// TwinCAT 3 PLC project PLC
// ProgramVersion: 3.1.4024.0
// libraries:
//   Tc2_EtherCAT, * (Beckhoff Automation GmbH)
//   Tc2_MC2, * (Beckhoff Automation GmbH)
//   Tc2_NC, * (Beckhoff Automation GmbH)
//   Tc2_Standard, * (Beckhoff Automation GmbH)
//   Tc2_System, * (Beckhoff Automation GmbH)
//   Tc2_Utilities, * (Beckhoff Automation GmbH)
//   Tc3_Module, * (Beckhoff Automation GmbH)
// project tree:
//   DUTs/EtherCAT_Diag/ E_EcDiacStatus.TcDUT, E_EcGetSlaveName.TcDUT, E_EcSystemStatus.TcDUT, ST_EcTerminalDiagInfo.TcDUT
//   DUTs/TwinSAFE_Diag/ ST_AdsAddr.TcDUT
//   DUTs/TwinSAFE_Diag/TwinSAFE_Connection/EL1904/ ST_TsConnectionInfoEL1904.TcDUT, ST_TsDiagObjectsBitsEL1904.TcDUT, ST_TsDiagObjectsEL1904.TcDUT, ST_TsSlaveInfoEL1904.TcDUT
//   DUTs/TwinSAFE_Diag/TwinSAFE_Connection/EL2904/ ST_TsConnectionInfoEL2904.TcDUT, ST_TsDiagObjectsBitsEL2904.TcDUT, ST_TsDiagObjectsEL2904.TcDUT, ST_TsSlaveInfoEL2904.TcDUT
//   DUTs/TwinSAFE_Diag/TwinSAFE_Connection/EL6910/ ST_TsDeviceInfoDataC.TcDUT, ST_TsSlaveInfoEL6910.TcDUT
//   DUTs/TwinSAFE_Diag/TwinSAFE_Connection/ E_TsCycleDiagObj.TcDUT, ST_TsConnectionInfo12Byte.TcDUT, ST_TsConnectionInfo1Byte.TcDUT, ST_TsConnectionInfo2Byte.TcDUT, ST_TsConnectionInfo4Byte.TcDUT, ST_TsConnectionInfo8Byte.TcDUT, ST_TsSlave2Temp.TcDUT, ST_TsSlave3Temp.TcDUT, ST_TsSlaveAddress.TcDUT, ST_TsSlaveAddressCRC.TcDUT
//   DUTs/TwinSAFE_Diag/TwinSAFE_Functionblocks/ E_TsFbType.TcDUT, ST_TsFbInfo.TcDUT
//   DUTs/TwinSAFE_Diag/TwinSAFE_Group/ ST_TsGroupInfo.TcDUT
//   GVLs/ IO.TcGVL
//   / PlcTask.TcTTO
//   POUs/ FB_EcGetSlaveName.TcPOU (not stored), FB_TwinSafeConnectionEL1904.TcPOU, FB_TwinSafeConnectionEL2904.TcPOU (not stored), FB_TwinSafeConnectionEL6910.TcPOU (not stored), FB_TwinSafeFB.TcPOU, FB_TwinSafeGroup.TcPOU, FB_TwinSafeGroupExt.TcPOU, F_Scale.TcPOU, MAIN.TcPOU, PRG_Safety.TcPOU
// real-time tasks:
//   TASK PlcTask: cycle T#10ms, priority 20, ADS port 350
// motion (NC):
//   TASK NC-Task 1 SAF: cycle T#2ms, priority 4, ADS port 501
//   TASK NC-Task 1 SVB: cycle T#10ms, priority 8, ADS port 511
//   AXIS Axis 1 (id 1)
//     OtherSettings: AllowMotionCmdToSlave=true
//     encoder EncType=4
//       EncPara: MaxCount=#x0000ffff
//         Inc: RefSoftSyncMask=#x0000ffff
//     drive DrvType=24
//       Analog: TorqueSetpointScale=10, ScaleFactorActTorque=0.1
//       TimeComp: TaskDelayCycles=1
//     controller CtrType=1
//       CtrPara: PriorControlFactor=1
//         Observer: BandWidth=20
//   AXIS Axis 2 (id 2)
//     Dynamic: Acceleration=12727.1, Deceleration=12727.1, Jerk=38181.3
//     Velo: RefSearch=84.8472746666667, RefSync=84.8472746666667, SlowManual=424.236373333333, FastManual=2545.41824, Fast=8484.72746666667, Maximum=8484.73
//     OtherSettings: AllowMotionCmdToSlave=true
//     encoder EncType=19
//       EncPara: ScaleFactorNumerator=104.8576, ScaleFactorDenominator=1048576, MaxCount=#xffffffff
//     drive DrvType=16
//       DrvPara: MaxCount=#xffffffff, DriveControlDWord=#x00020000
//         Analog: VeloReferenz=9333.20021333334, VeloScale=32, TorqueSetpointScale=10, ScaleFactorActTorque=0.1
//         TimeComp: TaskDelayCycles=1
//     controller CtrType=1
//       CtrPara: PriorControlFactor=1
//         PosDiffControl: Enable=false
//         Observer: BandWidth=20
// I/O:
//   DEVICE Device 1 (EtherCAT), AmsNetId 5.71.184.138.2.1
//     Term 1 (EK1200) [EK1200-5000 EtherCAT Power supply (2A E-Bus)]
//       Term 2 (EL1014) [EL1014 4Ch. Dig. Input 24V, 10µs]
//       Term 3 (EL2014) [EL2014 4Ch. Dig. Output 24V, 0,5A, Diagnostic]
//       Term 4 (EL6910) [EL6910, TwinSAFE PLC]
//       Term 5 (EL1904) [EL1904, 4 Ch. Safety Input 24V, TwinSAFE]
//         modules: Module 1 (FSOES)
//       Term 6 (EL3102) [EL3102 2Ch. Ana. Input +/-10V, Diff.]
//       Term 7 (EL9512) [EL9512 Power supply terminal 12V]
//       Term 8 (EK1122) [EK1122 2 port EtherCAT junction]
//         Term 9 (EK1818) [EK1818 EtherCAT IO-Coupler  (1A E-Bus, 8 Ch. Dig. In, 3ms, 4 Ch. Dig. Out 24V, 0,5A)]
//           Term 10 (EL1809) [EL1809 16Ch. Dig. Input 24V, 3ms]
//           Term 11 (EL2809) [EL2809 16Ch. Dig. Output 24V, 0.5A]
//           Term 12 (EL2904) [EL2904, 4 Ch. Safety Output 24V, 0.5A, TwinSAFE]
//             modules: Module 1 (FSOES), Module 2 (DO)
//           Term 13 (EL9110) [EL9110 Power Supplier with LED (24V, Diagnostics)]
//           Term 14 (EL7031) [EL7031 1Ch. Stepper motor output stage (24V, 1.5A)]
//           Term 15 (EL7201-9014) [EL7201-9014 1Ch. MDP742 Servo motor output stage with OCT (50V, 2.8A RMS) and STO input]
//           Term 33 (EL4102) [EL4102 2Ch. Ana. Output  0-10V, 16bit]
//           Term 35 (EL9011) [EL9011 End Terminal]
//       Term 16 (EK1110) [EK1110 EtherCAT extension]
// variable links:
//   Device 1 (EtherCAT) <-> Device 1 (EtherCAT)/Term 1 (EK1200)/Term 4 (EL6910)
//     Term 1 (EK1200)/Term 5 (EL1904)/Module 1 (FSOES)/RxPDO/FSOE <-> ConnectionInputs/TwinSafeGroup1.Term 5 (EL1904) - Module 1 (FSOES)_3 TxPDO
//     Term 1 (EK1200)/Term 8 (EK1122)/Term 9 (EK1818)/Term 12 (EL2904)/Module 1 (FSOES)/RxPDO/FSOE <-> ConnectionInputs/TwinSafeGroup1.Term 12 (EL2904) - Module 1 (FSOES)_4 TxPDO
//   Device 1 (EtherCAT) <-> Device 1 (EtherCAT)/Term 1 (EK1200)/Term 5 (EL1904)
//     Term 1 (EK1200)/Term 4 (EL6910)/ConnectionOutputs/TwinSafeGroup1.Term 5 (EL1904) - Module 1 (FSOES)_3 RxPDO <-> Module 1 (FSOES)/TxPDO/FSOE
//   Device 1 (EtherCAT) <-> Device 1 (EtherCAT)/Term 1 (EK1200)/Term 8 (EK1122)/Term 9 (EK1818)/Term 12 (EL2904)
//     Term 1 (EK1200)/Term 4 (EL6910)/ConnectionOutputs/TwinSafeGroup1.Term 12 (EL2904) - Module 1 (FSOES)_4 RxPDO <-> Module 1 (FSOES)/TxPDO/FSOE
//   NC-Task 1 SAF/Axes/Axis 1 <-> Device 1 (EtherCAT)/Term 1 (EK1200)/Term 8 (EK1122)/Term 9 (EK1818)/Term 14 (EL7031)
//     Drive/Inputs/In/nState1 @bit 3 <-> STM Status/Status/Error
//     Drive/Inputs/In/nState1 @bit 5 <-> STM Status/Status/Moving negative
//     Drive/Inputs/In/nState1 @bit 4 <-> STM Status/Status/Moving positive
//     Drive/Inputs/In/nState1 @bit 1 <-> STM Status/Status/Ready
//     Drive/Inputs/In/nState1 <-> STM Status/Status/Ready to enable
//     Drive/Inputs/In/nState1 @bit 6 <-> STM Status/Status/Torque reduced
//     Drive/Inputs/In/nState1 @bit 2 <-> STM Status/Status/Warning
//     Drive/Inputs/In/nState2 @bit 3 <-> STM Status/Status/Digital input 1
//     Drive/Inputs/In/nState2 @bit 4 <-> STM Status/Status/Digital input 2
//     Drive/Inputs/In/nState2 @bit 5 <-> STM Status/Status/Sync error
//     Drive/Inputs/In/nState2 @bit 7 <-> STM Status/Status/TxPDO Toggle
//     Drive/Inputs/In/nState4 @bit 1 <-> WcState/InputToggle
//     Drive/Inputs/In/nState4 <-> WcState/WcState
//     Drive/Outputs/Out/nCtrl1 <-> STM Control/Control/Enable
//     Drive/Outputs/Out/nCtrl1 @bit 2 <-> STM Control/Control/Reduce torque
//     Drive/Outputs/Out/nCtrl1 @bit 1 <-> STM Control/Control/Reset
//     Drive/Outputs/Out/nDataOut2[0] <-> STM Velocity/Velocity
//     Enc/Inputs/In/nDataIn1[0] <-> ENC Status compact/Counter value
//     Enc/Inputs/In/nDataIn2[0] <-> ENC Status compact/Latch value
//     Enc/Inputs/In/nState1 @bit 4 <-> ENC Status compact/Status/Counter overflow
//     Enc/Inputs/In/nState1 @bit 3 <-> ENC Status compact/Status/Counter underflow
//     Enc/Inputs/In/nState1 @bit 1 <-> ENC Status compact/Status/Latch extern valid
//     Enc/Inputs/In/nState1 @bit 2 <-> ENC Status compact/Status/Set counter done
//     Enc/Inputs/In/nState2 @bit 4 <-> ENC Status compact/Status/Status of extern latch
//     Enc/Inputs/In/nState2 @bit 5 <-> ENC Status compact/Status/Sync error
//     Enc/Inputs/In/nState2 @bit 7 <-> ENC Status compact/Status/TxPDO Toggle
//     Enc/Inputs/In/nState4 @bit 1 <-> WcState/InputToggle
//     Enc/Inputs/In/nState4 <-> WcState/WcState
//     Enc/Outputs/Out/nCtrl1 @bit 3 <-> ENC Control compact/Control/Enable latch extern on negative edge
//     Enc/Outputs/Out/nCtrl1 @bit 1 <-> ENC Control compact/Control/Enable latch extern on positive edge
//     Enc/Outputs/Out/nCtrl1 @bit 2 <-> ENC Control compact/Control/Set counter
//     Enc/Outputs/Out/nDataOut1[0] <-> ENC Control compact/Set counter value
//   NC-Task 1 SAF/Axes/Axis 2 <-> Device 1 (EtherCAT)/Term 1 (EK1200)/Term 8 (EK1122)/Term 9 (EK1818)/Term 15 (EL7201-9014)
//     Drive/Inputs/In/nDcOutputTime <-> InfoData/DcOutputShift
//     Drive/Inputs/In/nState1 <-> DRV Statusword/Statusword
//     Drive/Inputs/In/nState2 <-> DRV Statusword/Statusword @bit 8
//     Drive/Inputs/In/nState4 @bit 1 <-> WcState/InputToggle
//     Drive/Inputs/In/nState4 <-> WcState/WcState
//     Drive/Outputs/Out/nCtrl1 <-> DRV Controlword/Controlword
//     Drive/Outputs/Out/nCtrl2 <-> DRV Controlword/Controlword @bit 8
//     Drive/Outputs/Out/nDataOut2 <-> DRV Target velocity/Target velocity
//     Enc/Inputs/In/nDataIn1 <-> FB Position/Position
//     Enc/Inputs/In/nDcInputTime <-> InfoData/DcInputShift
//     Enc/Inputs/In/nState4 @bit 1 <-> WcState/InputToggle
//     Enc/Inputs/In/nState4 <-> WcState/WcState
//   PLC/PLC Instance <-> Device 1 (EtherCAT)/Term 1 (EK1200)/Term 2 (EL1014)
//     PlcTask Inputs/IO.bButton{1..4} <-> Channel {1..4}/Input  (4 links)
//   PLC/PLC Instance <-> Device 1 (EtherCAT)/Term 1 (EK1200)/Term 3 (EL2014)
//     PlcTask Outputs/IO.bLed{1..4} <-> DIG Outputs/Channel {1..4}/Output  (4 links)
//   PLC/PLC Instance <-> Device 1 (EtherCAT)/Term 1 (EK1200)/Term 4 (EL6910)
//     PlcTask Inputs/PRG_Safety.fbTsConnection_EL1904.stInfoData <-> Connection Info Data/TwinSafeGroup1.Term 5 (EL1904) - Module 1 (FSOES)_3 Info Data
//     PlcTask Inputs/PRG_Safety.fbTsConnection_EL2904.stInfoData <-> Connection Info Data/TwinSafeGroup1.Term 12 (EL2904) - Module 1 (FSOES)_4 Info Data
//     PlcTask Inputs/PRG_Safety.fbTsConnection_EL6910.nEcSlaveState <-> InfoData/State
//     PlcTask Inputs/PRG_Safety.fbTsConnection_EL6910.stEcAdsAddr <-> InfoData/AdsAddr
//     PlcTask Inputs/PRG_Safety.fbTsFB_Estop1.stInfoData <-> Function Block Info Data/TwinSafeGroup1.Network1.FBEstop1 Info Data
//     PlcTask Inputs/PRG_Safety.fbTsGroup_1.stInfoData <-> TwinSAFE Group Info Data/TwinSafeGroup1 Info Data
//     PlcTask Inputs/PRG_Safety.idiSerialnumber <-> Device Info Data/Serial Number
//     PlcTask Inputs/PRG_Safety.wProjectCrc <-> Device Info Data/Project CRC
//     PlcTask Outputs/PRG_Safety.ErrAck <-> StandardOutputs/Standard In Var 1
//     PlcTask Outputs/PRG_Safety.RunStop <-> StandardOutputs/Standard In Var 2
//   PLC/PLC Instance <-> Device 1 (EtherCAT)/Term 1 (EK1200)/Term 5 (EL1904)
//     PlcTask Inputs/PRG_Safety.fbTsConnection_EL1904.nEcSlaveState <-> InfoData/State
//     PlcTask Inputs/PRG_Safety.fbTsConnection_EL1904.stEcAdsAddr <-> InfoData/AdsAddr
//   PLC/PLC Instance <-> Device 1 (EtherCAT)/Term 1 (EK1200)/Term 6 (EL3102)
//     PlcTask Inputs/IO.nSpeedCmd <-> AI Standard Channel 1/Value
//   PLC/PLC Instance <-> Device 1 (EtherCAT)/Term 1 (EK1200)/Term 8 (EK1122)/Term 9 (EK1818)/Term 12 (EL2904)
//     PlcTask Inputs/PRG_Safety.fbTsConnection_EL2904.nEcSlaveState <-> InfoData/State
//     PlcTask Inputs/PRG_Safety.fbTsConnection_EL2904.stEcAdsAddr <-> InfoData/AdsAddr
//   PLC/PLC Instance <-> Device 1 (EtherCAT)/Term 1 (EK1200)/Term 8 (EK1122)/Term 9 (EK1818)/Term 33 (EL4102)
//     PlcTask Outputs/IO.nPotentiometer <-> Channel 2/Output
//   PLC/PLC Instance <-> NC-Task 1 SAF/Axes/Axis 2
//     PlcTask Inputs/MAIN.AxisB.NcToPlc <-> Outputs/ToPlc
//     PlcTask Outputs/MAIN.AxisB.PlcToNc <-> Inputs/FromPlc

CONFIGURATION PLC
    RESOURCE PLC ON TwinCAT3
        TASK PlcTask(INTERVAL := T#10ms, PRIORITY := 20);
        PROGRAM MAIN WITH PlcTask : MAIN;
    END_RESOURCE
END_CONFIGURATION

// ---- DUTs/EtherCAT_Diag/E_EcDiacStatus.TcDUT
TYPE E_EcDiacStatus :
(

	eEcDiac_Start							:= 0, 
	eEcDiac_Delay							,
	eEcDiac_ReadMasterState					,
	eEcDiac_ReadSlaveState

);
END_TYPE
(* End *)

// ---- DUTs/EtherCAT_Diag/E_EcGetSlaveName.TcDUT
TYPE E_EcGetSlaveName :
(

	eEcGetSlaveName_Start						:= 0,
	eEcGetSlaveName_Init						:= 10,
	eEcGetSlaveName_ReadAllSlaveAddr			:= 100,
	eEcGetSlaveName_ReadSlaveName				,
	eEcGetSlaveName_Done						:= 500,
	eEcGetSlaveName_ErrorStep 					:= 999,
	eEcGetSlaveName_NoError

);
END_TYPE
(* End *)

// ---- DUTs/EtherCAT_Diag/E_EcSystemStatus.TcDUT
TYPE E_EcSystemStatus :
(

	eEcSystem_Start							:= 0,
	eEcSystem_ReadConfSystem

);
END_TYPE
(* End *)

// ---- DUTs/EtherCAT_Diag/ST_EcTerminalDiagInfo.TcDUT
TYPE ST_EcTerminalDiagInfo :
STRUCT

	nAddr									:UINT;
	sType									:STRING(15);
	sName									:STRING(31);
	sTerminalStatus							:STRING(60);

END_STRUCT
END_TYPE
(* End *)

// ---- DUTs/TwinSAFE_Diag/ST_AdsAddr.TcDUT
TYPE ST_AdsAddr :
STRUCT

	netId									:AMSNETID;
	port									:WORD;

END_STRUCT
END_TYPE

// ---- DUTs/TwinSAFE_Diag/TwinSAFE_Connection/EL1904/ST_TsConnectionInfoEL1904.TcDUT
TYPE ST_TsConnectionInfoEL1904 :
(*******************************************************************************************************
Description			:	Connection information data of EtherCAT Slaves with 1 byte safe data 
Supported terminals : 	EL1904, EL2904...
Date 				:	04.04.2016
********************************************************************************************************)
STRUCT

	nState 	 								:USINT;
	nDiag 		 							:USINT;
	nInOutSafeDataByte1						:BYTE;
	
END_STRUCT
END_TYPE
(* End *)

// ---- DUTs/TwinSAFE_Diag/TwinSAFE_Connection/EL1904/ST_TsDiagObjectsBitsEL1904.TcDUT
TYPE ST_TsDiagObjectsBitsEL1904 :
(*******************************************************************************************************
Description			:	Index 16#800E Diagnostic objects
Supported terminals : 	EL1904
Documentation 		:	EL1904 TwinSAFE input terminal with 4 fail-safe inputs
Version/Date 		:	V1.5.2/02.10.2015
********************************************************************************************************)
STRUCT
	
(* Sensor test error *)
	bErrInput1								:BOOL;	(* Error input 1 - Bit0 - Error at input 1 *)
	bErrInput2								:BOOL;	(* Error input 2 - Bit1 - Error at input 2 *)
	bErrInput3								:BOOL;	(* Error input 3 - Bit2 - Error at input 3 *)
	bErrInput4								:BOOL;	(* Error input 4 - Bit3 - Error at input 4 *)

(* Error during two channel evaluation *)
	bErrFirstInputPair						:BOOL;	(* Error input 1..2 - Bit0 - Error in the first input pair *)
	bErrSecondInputPair						:BOOL;	(* Error input 3..4 - Bit1 - Error in the second input pair *)

(* Error in the safety mat operating mode: input pair disagree *)
	bMatOpModeErrFirstInputPair				:BOOL;	(* Error input 1..2 - Bit1, Bit0 - Mat operating mode - Error in the first input pair *)
	bMatOpModeErrSecondInputPair			:BOOL;	(* Error input 3..4 - Bit3, Bit2 - Mat operating mode - Error in the second input pair *)

(* Error in the safety mat operating mode: external supply *)
	bMatOpModeExtSupplyErrInput1			:BOOL;	(* Error input 1 - Bit0 - Mat operating mode external supply - Error at input 1 *)
	bMatOpModeExtSupplyErrInput2			:BOOL;	(* Error input 2 - Bit1 - Mat operating mode external supply - Error at input 2 *)
	bMatOpModeExtSupplyErrInput3			:BOOL;	(* Error input 3 - Bit2 - Mat operating mode external supply - Error at input 3 *)
	bMatOpModeExtSupplyErrInput4			:BOOL;	(* Error input 4 - Bit3 - Mat operating mode external supply - Error at input 4 *)
	
END_STRUCT
END_TYPE
(* End *)

// ---- DUTs/TwinSAFE_Diag/TwinSAFE_Connection/EL1904/ST_TsDiagObjectsEL1904.TcDUT
TYPE ST_TsDiagObjectsEL1904 :
(*******************************************************************************************************
Description			:	Index 16#800E Diagnostic objects
Supported terminals : 	EL1904
Documentation 		:	EL1904 TwinSAFE input terminal with 4 fail-safe inputs
Version/Date 		:	V1.5.2/02.10.2015
********************************************************************************************************)
STRUCT

	nDummyData1								:ARRAY[0..8] OF UINT;

(* Sensor test error *)
	nSensorTestError						:UINT;

(* Error during two channel evaluation *)
	nDuringTwoChannelEvaluationError		:UINT;

(* Error in the safety mat operating mode: input pair disagree *)
	nMatModeInputPairDisagreeError			:UINT;

(* Error in the safety mat operating mode: external supply *)
	nMatModeExternalSupplyError				:UINT;

	nDummyData2								:ARRAY[0..2] OF UINT;

END_STRUCT
END_TYPE
(* End *)

// ---- DUTs/TwinSAFE_Diag/TwinSAFE_Connection/EL1904/ST_TsSlaveInfoEL1904.TcDUT
TYPE ST_TsSlaveInfoEL1904 :
STRUCT

(* act_EcSlaveIdentify *)
	sEcSlaveType							:STRING(15);
	sEcSlaveName							:STRING(31) := '';
	bSlaveIdentify							:BOOL;
	bSlaveTypeError							:BOOL;

	stTsSlaveAddress 						:ST_TsSlaveAddress;
	bSlaveAddressOk							:BOOL;

	nEcSlaveFSoEAddr						:UINT;
	nEcSlaveSerialNumber					:UDINT;

(* act_ConnectionState *)
	sState									:STRING;
	
(* act_ConnectionDiag *)
	sDiag									:STRING;
	sFault									:STRING;						(* FailSafe Error (Hardware)*)
	bError									:BOOL;							(* TwinSAFE-Error *)

(* act_ReadDiagObjects *)
	stSlaveTemp								:ST_TsSlave2Temp;
	bIntTempWarning1						:BOOL;							(* Temperature warning: T1 *)
	bIntTempWarning2						:BOOL;							(* Temperature warning: T2 *)
	stTsDiagObjectsBitsEL1904				:ST_TsDiagObjectsBitsEL1904;

	
(* act_Signals *)
	bChannel1								:BOOL;							
	bChannel2								:BOOL;
	bChannel3								:BOOL;
	bChannel4								:BOOL;

END_STRUCT
END_TYPE
(* End *)

// ---- DUTs/TwinSAFE_Diag/TwinSAFE_Connection/EL2904/ST_TsConnectionInfoEL2904.TcDUT
TYPE ST_TsConnectionInfoEL2904 :
(*******************************************************************************************************
Description			:	Connection information data of EtherCAT Slaves with 1 byte safe data 
Supported terminals : 	EL1904, EL2904...
Date 				:	04.04.2016
********************************************************************************************************)
STRUCT

	nState 	 								:USINT;
	nDiag 		 							:USINT;
	nInOutSafeDataByte1						:BYTE;
	
END_STRUCT
END_TYPE
(* End *)

// ---- DUTs/TwinSAFE_Diag/TwinSAFE_Connection/EL2904/ST_TsDiagObjectsBitsEL2904.TcDUT
TYPE ST_TsDiagObjectsBitsEL2904 :
(*******************************************************************************************************
Description			:	Index 16#800E Diagnostic objects
Supported terminals : 	EL2904
Documentation 		:	EL2904 TwinSAFE output terminal with 4 fail-safe outputs
Version/Date 		:	V1.6.2/02.10.2015
********************************************************************************************************)
STRUCT
	
(* Error at the outputs *)
	bEsOrCcErrOutput1						:BOOL;	(* Error output 1 - Bit0 - External supply or cross circuit *)
	bEsOrCcErrOutput2						:BOOL;	(* Error output 2 - Bit1 - External supply or cross circuit *)
	bEsOrCcErrOutput3						:BOOL;	(* Error output 3 - Bit2 - External supply or cross circuit *)
	bEsOrCcErrOutput4						:BOOL;	(* Error output 4 - Bit3 - External supply or cross circuit *)
	bOlOrCvErrOutput1						:BOOL;	(* Error output 1 - Bit4 - Open load or current below minimum value of 20 mA or current above maximum value of 500mA *)
	bOlOrCvErrOutput2						:BOOL;	(* Error output 2 - Bit5 - Open load or current below minimum value of 20 mA or current above maximum value of 500mA *)
	bOlOrCvErrOutput3						:BOOL;	(* Error output 3 - Bit6 - Open load or current below minimum value of 20 mA or current above maximum value of 500mA *)
	bOlOrCvErrOutput4						:BOOL;	(* Error output 4 - Bit7 - Open load or current below minimum value of 20 mA or current above maximum value of 500mA *)

(* Supply error *)
	bFieldVoltageTooHigh					:BOOL;	(* Supply error - Bit 0 - Field voltage too high *)
	bFieldVoltageTooLow						:BOOL;	(* Supply error - Bit 1 - Field voltage too low *)

(* Temperature error *)
	nOvertemperatureC1						:BOOL;	(* Temperature error - Bit 0 - Overtemperature µC1 *)
	nOvertemperatureC2						:BOOL;	(* Temperature error - Bit 1 - Overtemperature µC2 *)
	nOvertemperatureOutputs					:BOOL;	(* Temperature error - Bit 2 - Overtemperature of the output board *)
	nTemperatureTooLowC1					:BOOL;	(* Temperature error - Bit 3 - Temperature too low µC1 *)
	nTemperatureTooLowC2					:BOOL;	(* Temperature error - Bit 4 - Temperature too low µC2 *)
	nTemperatureTooLowOutputs				:BOOL;	(* Temperature error - Bit 5 - Temperature of the output board too low *)
	nOvertemperatureDiffBoard				:BOOL;	(* Temperature error - Bit 6 - Temperature difference on the processor board too large *)
	nOvertemperatureDiffBetwBoards			:BOOL;	(* Temperature error - Bit 7 - Temperature difference between the boards is too large *)
	
END_STRUCT
END_TYPE
(* End *)

// ---- DUTs/TwinSAFE_Diag/TwinSAFE_Connection/EL2904/ST_TsDiagObjectsEL2904.TcDUT
TYPE ST_TsDiagObjectsEL2904 :
(*******************************************************************************************************
Description			:	Index 16#800E Diagnostic objects
Supported terminals : 	EL2904
Documentation 		:	EL2904 TwinSAFE output terminal with 4 fail-safe outputs
Version/Date 		:	V1.6.2/02.10.2015
********************************************************************************************************)
STRUCT
	
	nDummyData1								:ARRAY[0..10] OF UINT;

(* Error at the outputs *)
	nErrorOutputs							:UINT;

(* Supply error *)
	nSupplyError							:UINT;

(* Temperature error *)
	nTemperatureError						:UINT;

	nDummyData2								:ARRAY[0..1] OF UINT;

END_STRUCT
END_TYPE
(* End *)

// ---- DUTs/TwinSAFE_Diag/TwinSAFE_Connection/EL2904/ST_TsSlaveInfoEL2904.TcDUT
TYPE ST_TsSlaveInfoEL2904 :
STRUCT

(* act_EcSlaveIdentify *)
	sEcSlaveType							:STRING(15);
	sEcSlaveName							:STRING(31) := '';
	bSlaveIdentify							:BOOL;
	bSlaveTypeError							:BOOL;

	stTsSlaveAddress 						:ST_TsSlaveAddress;
	bSlaveAddressOk							:BOOL;	
	
	nEcSlaveFSoEAddr						:UINT;
	nEcSlaveSerialNumber					:UDINT;
	
(* act_ConnectionState *)
	sState									:STRING;
	
(* act_ConnectionDiag *)
	sDiag									:STRING;
	sFault									:STRING(255);					(* FailSafe Error (Hardware)*)
	bError									:BOOL;							(* TwinSAFE-Error *)

(* act_ReadDiagObjects *)
	stSlaveTemp								:ST_TsSlave3Temp;
	bIntTempWarning1						:BOOL;							(* Temperature warning: T1 *)
	bIntTempWarning2						:BOOL;							(* Temperature warning: T2 *)
	bWarningLevelTempOutputs				:BOOL;							(* Temperature 2 [°C] *)
	stTsDiagObjectsBitsEL2904				:ST_TsDiagObjectsBitsEL2904;
	
(* act_Signals *)
	bChannel1								:BOOL;							
	bChannel2								:BOOL;
	bChannel3								:BOOL;
	bChannel4								:BOOL;	

END_STRUCT
END_TYPE
(*End*)

// ---- DUTs/TwinSAFE_Diag/TwinSAFE_Connection/EL6910/ST_TsDeviceInfoDataC.TcDUT
TYPE ST_TsDeviceInfoDataC :
(*******************************************************************************************************
Description			:	EtherCAT master terminals device info controller
Supported terminals : 	EL6910
Date 				:	25.05.2018
********************************************************************************************************)
STRUCT

	nVoltageC						:UINT;	(* Voltage controller [mV] *)
	nTemperatureC					:INT;	(* Temperature controller [°C] *)
	FirmwareCRC						:UINT;	(**)
	VendordataCRC					:UINT;	(**)
END_STRUCT
END_TYPE
(* End *)

// ---- DUTs/TwinSAFE_Diag/TwinSAFE_Connection/EL6910/ST_TsSlaveInfoEL6910.TcDUT
TYPE ST_TsSlaveInfoEL6910 :
STRUCT

(* act_EcSlaveIdentify *)
	sEcSlaveType							:STRING(15);
	sEcSlaveName							:STRING(31) := '';
	bSlaveIdentify							:BOOL;
	bSlaveTypeError							:BOOL;	
	{attribute 'displaymode':='hex'}
	nEcSlaveProjectCRC						:UINT;
	
	stTsSlaveAddress 						:ST_TsSlaveAddressCRC;
	bSlaveAddressOk							:BOOL;
	
	nEcSlaveFSoEAddr						:UINT;
	nEcSlaveSerialNumber					:UDINT;
	
(* act_ReadDiagObjects *)
	stDeviceInfoDataC1						:ST_TsDeviceInfoDataC;
	stDeviceInfoDataC2						:ST_TsDeviceInfoDataC;
	bIntTempWarning1						:BOOL;							(* Temperature warning: T1 *)
	bIntTempWarning2						:BOOL;							(* Temperature warning: T2 *)

END_STRUCT
END_TYPE

// ---- DUTs/TwinSAFE_Diag/TwinSAFE_Connection/E_TsCycleDiagObj.TcDUT
TYPE E_TsCycleDiagObj :
(*******************************************************************************************************
Description			:	Enumeration read diagnosis objects steps 
Supported terminals : 	EL1904, EL2904, EL69xx, AX5805, AX5806
Date 				:	04.04.2016
********************************************************************************************************)
(

	eCycleDiagObj_Init						:= 0,
	eCycleDiagObj_ReadTemperature			,
	eCycleDiagObj_ReadTemperatureC1			,
	eCycleDiagObj_ReadTemperatureC2			,
	eCycleDiagObj_ReadErrorIndices			,	
	eCycleDiagObj_ReadDiag					,	
	eCycleDiagObj_ReadDelay					,	
	eCycleDiagObj_Done						,
	eCycleDiagObj_Error						:=999,
	eCycleDiagObj_NoError					
	
);
END_TYPE
(* End *)

// ---- DUTs/TwinSAFE_Diag/TwinSAFE_Connection/ST_TsConnectionInfo12Byte.TcDUT
TYPE ST_TsConnectionInfo12Byte :
(*******************************************************************************************************
Description			:	Connection information data of EtherCAT Slaves with 12 byte safe data   
Supported terminals : 	EK1960
Date 				:	04.11.2018
********************************************************************************************************)
STRUCT

	nState  								:USINT;
	nDiag 	 								:USINT;
	
	nInOutSafeDataByte1	 					:BYTE;
	nInOutSafeDataByte2	 					:BYTE;
	nInOutSafeDataByte3	 					:BYTE;
	nInOutSafeDataByte4 					:BYTE;
	nInOutSafeDataByte5 					:BYTE;
	nInOutSafeDataByte6 					:BYTE;
	nInOutSafeDataByte7 					:BYTE;
	nInOutSafeDataByte8 					:BYTE;
	nInOutSafeDataByte9 					:BYTE;
	nInOutSafeDataByte10					:BYTE;
	nInOutSafeDataByte11					:BYTE;
	nInOutSafeDataByte12					:BYTE;

END_STRUCT
END_TYPE
(* End *)

// ---- DUTs/TwinSAFE_Diag/TwinSAFE_Connection/ST_TsConnectionInfo1Byte.TcDUT
TYPE ST_TsConnectionInfo1Byte :
(*******************************************************************************************************
Description			:	Connection information data of EtherCAT Slaves with 1 byte safe data 
Supported terminals : 	EL1904, EL2904...
Date 				:	04.04.2016
********************************************************************************************************)
STRUCT

	nState 	 								:USINT;
	nDiag 		 							:USINT;
	nInOutSafeDataByte1						:BYTE;
	
END_STRUCT
END_TYPE
(* End *)

// ---- DUTs/TwinSAFE_Diag/TwinSAFE_Connection/ST_TsConnectionInfo2Byte.TcDUT
TYPE ST_TsConnectionInfo2Byte :
(*******************************************************************************************************
Description			:	Connection information data of EtherCAT Slaves with 2 byte safe data 
Supported terminals : 	EK1914...
Date 				:	04.04.2016
********************************************************************************************************)
STRUCT

	nState 	 								:USINT;
	nDiag 		 							:USINT;
	nInOutSafeDataByte1						:BYTE;
	nInOutSafeDataByte2						:BYTE;
	
END_STRUCT
END_TYPE
(* End *)

// ---- DUTs/TwinSAFE_Diag/TwinSAFE_Connection/ST_TsConnectionInfo4Byte.TcDUT
TYPE ST_TsConnectionInfo4Byte :
(*******************************************************************************************************
Description			:	Connection information data of EtherCAT Slaves with 2 byte input and 2 byte output safe data  
Supported terminals : 	EP1957
Date 				:	04.11.2018
********************************************************************************************************)
STRUCT

	nState  								:USINT;
	nDiag 	 								:USINT;
	nInOutSafeDataByte1						:BYTE;
	nInOutSafeDataByte2						:BYTE;
	nInOutSafeDataByte3						:BYTE;
	nInOutSafeDataByte4						:BYTE;

END_STRUCT
END_TYPE
(* End *)

// ---- DUTs/TwinSAFE_Diag/TwinSAFE_Connection/ST_TsConnectionInfo8Byte.TcDUT
TYPE ST_TsConnectionInfo8Byte :
(*******************************************************************************************************
Description			:	Connection information data of EtherCAT Slaves with 4 byte input and 4 byte output safe data  
Supported terminals : 	AX5805(2 Axis)
Date 				:	04.11.2018
********************************************************************************************************)
STRUCT

	nState  								:USINT;
	nDiag 	 								:USINT;
	nInOutSafeDataByte1						:BYTE;
	nInOutSafeDataByte2						:BYTE;
	nInOutSafeDataByte3						:BYTE;
	nInOutSafeDataByte4						:BYTE;
	nInOutSafeDataByte5 					:BYTE;
	nInOutSafeDataByte6 					:BYTE;
	nInOutSafeDataByte7 					:BYTE;
	nInOutSafeDataByte8 					:BYTE;

END_STRUCT
END_TYPE
(* End *)

// ---- DUTs/TwinSAFE_Diag/TwinSAFE_Connection/ST_TsSlave2Temp.TcDUT
TYPE ST_TsSlave2Temp :
(*******************************************************************************************************
Description			:	EtherCAT Slaves with 2 internal temperatures
Supported terminals : 	EL1904, AX5805, AX5806
Date 				:	04.04.2016
********************************************************************************************************)
STRUCT

	nInternalTemperature1				:INT;	(* Temperature 1 [°C] *)
	nInternalTemperature2				:INT;	(* Temperature 2 [°C] *)
	
END_STRUCT
END_TYPE
(* End *)

// ---- DUTs/TwinSAFE_Diag/TwinSAFE_Connection/ST_TsSlave3Temp.TcDUT
TYPE ST_TsSlave3Temp :
(*******************************************************************************************************
Description			:	EtherCAT Slaves with 3 internal temperatures
Supported terminals : 	EL2904
Date 				:	04.04.2016
********************************************************************************************************)
STRUCT
	
	nInternalTemperature1					:INT;	(* Temperature 1 [°C] *)
	nInternalTemperature2					:INT;	(* Temperature 2 [°C] *)
	nInternalTemperatureOutputs				:INT;	(* Temperature 2 [°C] *)
	
END_STRUCT
END_TYPE
(* End *)

// ---- DUTs/TwinSAFE_Diag/TwinSAFE_Connection/ST_TsSlaveAddress.TcDUT
TYPE ST_TsSlaveAddress :
(*******************************************************************************************************
Description			:	EtherCAT Slaves Address information
Supported terminals : 	EL1904, EL2904
Date 				:	25.05.2018
********************************************************************************************************)
STRUCT

	nEcSlaveFSoEAddr						:UINT;
	nEcSlaveSerialNumber					:ARRAY[0..1] OF WORD;

END_STRUCT
END_TYPE
(* End *)

// ---- DUTs/TwinSAFE_Diag/TwinSAFE_Connection/ST_TsSlaveAddressCRC.TcDUT
TYPE ST_TsSlaveAddressCRC :
(*******************************************************************************************************
Description			:	EtherCAT Slaves Address information
Supported terminals : 	EL6900, EL6910
Date 				:	25.05.2018
********************************************************************************************************)
STRUCT

	nEcSlaveFSoEAddr						:UINT;
	nEcSlaveSerialNumber					:ARRAY[0..1] OF WORD;
	nEcSlaveProjectCRC						:UINT;

END_STRUCT
END_TYPE
(* End *)

// ---- DUTs/TwinSAFE_Diag/TwinSAFE_Functionblocks/E_TsFbType.TcDUT
TYPE E_TsFbType :
(*******************************************************************************************************
Description			:	Enumeration TwinSAFE function block list
Documentation 		:	TwinSAFE-Logik-FB TwinCAT function blocks for TwinSAFE logic terminals
Supported hardware	: 	KL6904 / EL6900 / EL6910 / EJ6910 / EK1960
Version/Date 		:	V3.1.0/26.10.2016
********************************************************************************************************)
(
	
(* KL6904 / EL6900 / EL6910 / EJ6910 / EK1960 *)
	FB_TYPE_AND								:=0,
	FB_TYPE_OR								,
	FB_TYPE_OPMODE							,
	FB_TYPE_ESTOP							,
	FB_TYPE_MON								,
	FB_TYPE_DECOUPLER						,
	FB_TYPE_TWOHAND							,
	FB_TYPE_MUTING							,
	FB_TYPE_EDM								,
	FB_TYPE_RS								,
	FB_TYPE_SR								,
	FB_TYPE_TON								,
	FB_TYPE_TOF								,
	FB_TYPE_CONSHUT							,
(* only EL6910 / EJ6910 / EK1960 *)
	FB_TYPE_ADD								,
	FB_TYPE_SUB								,
	FB_TYPE_MUL								,
	FB_TYPE_DIV								,
	FB_TYPE_COMPARE							,
	FB_TYPE_LIMIT							,
	FB_TYPE_COUNTER							,
	FB_TYPE_SCALE							,
	FB_TYPE_SPEED							,
	FB_TYPE_LOADSENSING						,
	FB_TYPE_CAMMONITOR						,
	FB_TYPE_SLI								,
	FB_TYPE_ENVELOPE						,
	FB_TYPE_VIOLATIONCOUNTER				

);
END_TYPE
(* End *)

// ---- DUTs/TwinSAFE_Diag/TwinSAFE_Functionblocks/ST_TsFbInfo.TcDUT
TYPE ST_TsFbInfo :
STRUCT
	
	nState  								:USINT;
	nDiag  									:UINT;

END_STRUCT
END_TYPE
(* End *)

// ---- DUTs/TwinSAFE_Diag/TwinSAFE_Group/ST_TsGroupInfo.TcDUT
TYPE ST_TsGroupInfo :
STRUCT

	nState	 	 							:USINT;
	nDiag 	 								:USINT;

END_STRUCT
END_TYPE
(* End *)

// ---- GVLs/IO.TcGVL
{attribute 'qualified_only'}
VAR_GLOBAL
	bButton1 AT %I* : BOOL;
	bButton2 AT %I* : BOOL;
	bButton3 AT %I* : BOOL;
	bButton4 AT %I* : BOOL;
	bLed1 AT %Q* : BOOL;
	bLed2 AT %Q* : BOOL;
	bLed3 AT %Q* : BOOL;
	bLed4 AT %Q* : BOOL;
	nSpeedCmd AT %I* : INT;
	nPotentiometer AT %Q* : INT;
END_VAR

// ---- POUs/MAIN.TcPOU
PROGRAM MAIN
VAR
	nServoSpeed : DINT;
	
	AxisB : AXIS_REF;
	bSafetyCondition: BOOL;
	McPower : MC_Power;
	McReset : MC_Reset;
	McJogging : MC_Jog;
	McVelo : MC_MoveVelocity;
	McStop : MC_Stop;
	bVirtualMoveVelo : BOOL;
	bVirtualStop : BOOL;
	
	
	iState : INT; // my state
	nLastThrottle : INT;
END_VAR

bSafetyCondition:= PRG_Safety.fbTsConnection_EL2904.stTsSlaveInfo.bChannel1;

IF (IO.bButton1 OR bVirtualMoveVelo) AND bSafetyCondition THEN
	IO.bLed1:= TRUE;
END_IF

IF (IO.bButton2 OR bVirtualStop) OR NOT bSafetyCondition THEN
	IO.bLed1:=FALSE;
END_IF

IO.nPotentiometer := IO.nSpeedCmd;
nServoSpeed := F_Scale(nAIn:= IO.nSpeedCmd, 100.0, 2800.0, 0, 32767);

// Drive Control
AxisB.ReadStatus();
McPower(Axis:=AxisB,Enable:= TRUE, Enable_Positive:= TRUE, Enable_Negative:=TRUE);
McReset(Axis:=AxisB);
McJogging(Axis:=AxisB);

CASE iState OF
	0:
		iState:= 10; //initial
	10: // Start drive reset
		IF McPower.Status THEN
			McReset(Axis:= AxisB, Execute:=TRUE);
			IF McReset.Done THEN
				iState:=20;
			ELSIF McReset.Error THEN
				iState:=-999;		
			END_IF
		END_IF
			
	20: // Wait for drive to reset
		IF McPower.Status THEN
			iState:=30;
		END_IF
	30: // Wait for drive command
		//McJogging(Axis:=AxisB, JogForward := IO.bLed1);
		McVelo(
			Axis:= AxisB,
			Execute:= IO.bLed1 AND IO.nSpeedCmd <> nLastThrottle,
			Velocity:= nServoSpeed,
			Acceleration := 10000,
			Deceleration := 10000,
			Jerk := 10000000,
			Direction:= MC_DIRECTION.MC_Positive_Direction
		);
		IF NOT IO.bLed1 OR NOT bSafetyCondition THEN
			McVelo(Axis:=AxisB, Execute:= FALSE);
			iState:=900;
		END_IF
		nLastThrottle := IO.nSpeedCmd;
	900: // Stop Servo
		McStop(Axis:= AxisB, Execute:= TRUE);
		IF IO.bLed1 AND bSafetyCondition THEN
			McStop(Axis:= AxisB, Execute:= FALSE);
			iState:=30;
		END_IF
	-999: // Handle error
END_CASE


PRG_Safety();

END_PROGRAM

// ---- POUs/PRG_Safety.TcPOU
PROGRAM PRG_Safety
VAR
	ErrAck AT %Q* 	: BOOL;
	RstEstop AT %Q* : BOOL;
	RunStop AT %Q* 	: BOOL;
	ComErr AT %I* 	: BOOL;
	FbErr AT %I* 	: BOOL;
	OutErr AT %I* 	: BOOL;
	
	a : R_TRIG;
	ncounter:INT:=0;
	
	//=== TwinSAFE Diagnostic ===//
	// target system
		wProjectCrc 	AT %I*	: WORD;
		idiSerialnumber AT %I* 	: UDINT;
	//Group 1
		fbTsGroup_1			: FB_TwinSafeGroupExt;
		stTsGroupInfo		: ST_TsGroupInfo;
	//TwinSAFE Connection
		fbTsConnection_EL6910	: FB_TwinSafeConnectionEL6910;
		fbTsConnection_EL1904	: FB_TwinSafeConnectionEL1904;
		fbTsConnection_EL2904	: FB_TwinSafeConnectionEL2904;
	//Twinsafe function block
		fbTsFB_Estop1			: FB_TwinSafeFB;
	
END_VAR

a(CLK:=IO.bButton4 , Q=> );
IF a.Q THEN
	ncounter:=ncounter+1;
	IF ncounter >1 THEN
		ncounter:=0;
		IO.bLed2:= TRUE;

	END_IF
END_IF

IF ncounter = 1 THEN
	RunStop:=TRUE;
	IO.bLed2:= TRUE;

ELSE 
	RunStop:=FALSE;
	IO.bLed2:= FALSE;
END_IF

//Diagnostic
//TwinSAFE (Group 1)
fbTsGroup_1(
	bRun:= IO.bButton4, 
	bErrAck:= ErrAck, 
	sName:= 'Gr01_Estop');
//TwinSAFE connection
fbTsConnection_EL6910(tCoEReadCycle :=T#2S);
fbTsConnection_EL1904(tCoEReadCycle	:=T#2S) ;
fbTsConnection_EL2904(tCoEReadCycle	:=T#2S);
//Twinsafe Function Block
fbTsFB_Estop1(
	sName:= 'FBEstop1', 
	eFBType:= E_TsFbType.FB_TYPE_ESTOP, 
	nFbId:= 1);

END_PROGRAM

// ---- POUs/FB_TwinSafeGroupExt.TcPOU

FUNCTION_BLOCK FB_TwinSafeGroupExt
(*******************************************************************************************************
Description			:	Entries of the status and diagnostic TwinSAFE groups
ocumentation 		:	TwinSAFE-Logik-FB TwinCAT function blocks for TwinSAFE logic terminals
Supported hardware	: 	EL6910 / EJ6910 / EK1960
Version/Date 		:	V3.1.0/26.10.2016
********************************************************************************************************)
VAR_INPUT

	bRun							AT %Q*	:BOOL;				(* TwinSAFE group run - linked with the associated TwinSAFE Group in the TwinSAFE projekt *)
	bErrAck							AT %Q*	:BOOL;				(* TwinSAFE group error acknowledge - linked with the associated TwinSAFE Group in the TwinSAFE projekt *)
	sName									:STRING;			(* TwinSAFE group name *)

END_VAR
VAR_OUTPUT

	stInfoData						AT %I*	:ST_TsGroupInfo;	(* TwinSAFE Group Info Data *)
	bComErr							AT %I*	:BOOL;				(* TwinSAFE group communication error - linked with the associated TwinSAFE Group in the TwinSAFE projekt *)
	bFbErr							AT %I*	:BOOL;				(* TwinSAFE group function block error - linked with the associated TwinSAFE Group in the TwinSAFE projekt *)
	bOtherErr						AT %I*	:BOOL;				(* ModuleFault or AnalogValueFault or WaitComTimeoutFault *)
	bComStartUp						AT %I*	:BOOL;				(* At least one of the Connection of this group is in the StartUp *)
	bFbDeactive						AT %I*	:BOOL;				(* TwinSAFE group was deactivated *)
	bFbRun							AT %I*	:BOOL;				(* All Fbs are in run state *)
	bInRun							AT %I*	:BOOL;				(* TwinSAFE group is in run *)
	sState									:STRING;
	sDiag									:STRING;

END_VAR
VAR
END_VAR
(* End *)

(* TwinSAFE group status and diagnostic *)

(* THIS CODE IS ONLY AN EXAMPLE - YOU HAVE TO CHECK APTITUDE FOR YOUR APPLICATION *)

	CASE stInfoData.nState OF
		1:	sState := 'RUN';
		2:	sState := 'STOP';
		4:	sState := 'ERROR';
		5:	sState := 'RESET';
		6:	sState := 'START';
		7:	sState := 'STOPERROR';
		16:	sState := 'DEACTIVE';
		17:	sState := 'WAITCOMERROR';
	ELSE
		sState := 'undefined';
	END_CASE
	
	CASE stInfoData.nDiag OF
		0:	sDiag := 'No error';
		1:	sDiag := 'Fb error';
		2:	sDiag := 'Com error';
		3:	sDiag := 'Module error';
		4:	sDiag := 'CMP error';
		5:	sDiag := 'Deactivate error';
		6:	sDiag := 'Restart error';
	ELSE
		sDiag := 'undefined';
	END_CASE
	
(* End *)

END_FUNCTION_BLOCK

// ---- POUs/FB_TwinSafeConnectionEL1904.TcPOU
FUNCTION_BLOCK FB_TwinSafeConnectionEL1904
(*******************************************************************************************************
Description			:	Evaluate a TwinSAFE connection status and diagnosis to an EtherCAT terminal
Supported terminals : 	EL1904
Documentation 		:	EL1904 TwinSAFE input terminal with 4 fail-safe inputs
Version/Date 		:	V1.5.2/02.10.2015
Required libraries 	: 	TcSystem.lib (Tc2_System), TcEtherCAT.lib (Tc2_EtherCAT)
********************************************************************************************************)
VAR_INPUT
	
	tCoEReadCycle							:TIME 	:= T#0MS;				(* Read cycle CoE-Data, e.g. temperature *)

END_VAR
VAR_OUTPUT

	stInfoData						AT %I*	:ST_TsConnectionInfoEL1904;		(* [TwinSAFE logic] e.g. EL69xx \ Connection Info Data \ [Path] Info Data*)
	nEcSlaveState					AT %I*	:UINT ;							(* EL1904 \ InfoData \ State *)
	stEcAdsAddr						AT %I*	:ST_AdsAddr;					(* EL1904 \ InfoData \ AdsAddr *)

	stTsSlaveInfo							:ST_TsSlaveInfoEL1904;	
	
END_VAR
VAR

(* act_ConnectionDiag *)
	nDiag0_3								:BYTE;

(* act_ReadDiagObjects *)
	eReadDiagObjState						:E_TsCycleDiagObj;
	eReadDiagObjErrStep						:E_TsCycleDiagObj := E_TsCycleDiagObj.eCycleDiagObj_NoError;
	bReadDiagObjError						:BOOL;							(* Error in the diagnosis objects read cycle *)  
	bReadDiagObjReset						:BOOL;							(* Reset the diagnosis objects read cycle error *)
	fbTimer									:TON;
	fbEcCoeSdoRead							:FB_EcCoESdoReadEx;
	stDiagObjects							:ST_TsDiagObjectsEL1904;

(* act_EcSlaveIdentify *)
	fbEcGetSlaveName						:FB_EcGetSlaveName;

END_VAR
VAR CONSTANT
	
(* act_ReadDiagObjects *)
	nWarningLevelTemp1						:INT	:= 85;					(* Temperature 1 warning level [°C] *)
	nWarningLevelTemp2						:INT	:= 85;					(* Temperature 2 warning level [°C] *)

END_VAR
(* End *)

(* Function Block TwinSAFE connection status and diagnosis for EL1904 Terminals *)

(* THIS CODE IS ONLY AN EXAMPLE - YOU HAVE TO CHECK APTITUDE FOR YOUR APPLICATION *)

	(* Identify the EtherCAT slave *)
		act_EcSlaveIdentify();

	(* Evaluate the connection state *)
		act_ConnectionState();
	
	(* Evaluate the connection diagnosis *)
		act_ConnectionDiag();
	
	(* Evaluate the signals *)
		act_Signals();
	
	(* Evaluate the Terminal temperatures and diagnostic objects *)
		IF stTsSlaveInfo.bSlaveIdentify
			AND stTsSlaveInfo.bSlaveAddressOk
		THEN
			act_ReadDiagObjects();
		ELSE
			eReadDiagObjState := E_TsCycleDiagObj.eCycleDiagObj_Init;
		END_IF
		
(* End *)

ACTION act_ConnectionDiag:
(* Evaluate the connection diagnosis *)

	(* Evaluate Bit 0..3 *)
	nDiag0_3 := USINT_TO_BYTE(stInfoData.nDiag) AND 16#0F;

	CASE nDiag0_3 OF
		0:		stTsSlaveInfo.sDiag := 'No error';
		1:		stTsSlaveInfo.sDiag := 'Invalid command';
		2:		stTsSlaveInfo.sDiag := 'Unknown command';
		3:		stTsSlaveInfo.sDiag := 'Invalid connection ID';
		4:		stTsSlaveInfo.sDiag := 'Invalid CRC';
		5:		stTsSlaveInfo.sDiag := 'Watchdog time elapsed';
		6:		stTsSlaveInfo.sDiag := 'Invalid FSOE address';
		7:		stTsSlaveInfo.sDiag := 'Invalid data';
		8:		stTsSlaveInfo.sDiag := 'Invalid communication parameter length';
		9:		stTsSlaveInfo.sDiag := 'Invalid communication parameters';
		10:		stTsSlaveInfo.sDiag := 'Invalid user parameter length';
		11:		stTsSlaveInfo.sDiag := 'Invalid user parameter';
		12:		stTsSlaveInfo.sDiag := 'FSoE master reset';
		13:		stTsSlaveInfo.sDiag := 'Module err detected on slave, with option "Module error is ComError" activated';
		14:		stTsSlaveInfo.sDiag := 'Module err detected on EL290x, with option "Error acknowledge active" activated';
		15:		stTsSlaveInfo.sDiag := 'Slave not yet started, or unexpected error argument';
	END_CASE

	(* Evaluate Bit 4..7 *)
	stTsSlaveInfo.sFault:='';

	IF stInfoData.nDiag.4 
	THEN
		stTsSlaveInfo.sFault := 'FSoE slave error detected - '; 
	END_IF

	IF stInfoData.nDiag.5 
	THEN
		stTsSlaveInfo.sFault := concat(stTsSlaveInfo.sFault,'FSoE slave reports Failsafe Value active - ');
	END_IF

	IF stInfoData.nDiag.6 
	THEN
		stTsSlaveInfo.sFault := concat(stTsSlaveInfo.sFault,'StartUp - ');
	END_IF

	IF stInfoData.nDiag.7 
	THEN
		stTsSlaveInfo.sFault := concat(stTsSlaveInfo.sFault, 'FSoE master reports Failsafe Value active');
	END_IF
		
	(* Error *)
	stTsSlaveInfo.bError := stInfoData.nDiag <> 0;

(* End *)
END_ACTION

ACTION act_ConnectionState:
(* Evaluate the connection state *)

	CASE stInfoData.nState OF
		100:	stTsSlaveInfo.sState := 'Reset state';
		101:	stTsSlaveInfo.sState := 'Session state';
		102:	stTsSlaveInfo.sState := 'Connection state';
		103:	stTsSlaveInfo.sState := 'Parameter state';
		104:	stTsSlaveInfo.sState := 'Data state';
		105:	stTsSlaveInfo.sState := 'Shutdown state';
	ELSE
		stTsSlaveInfo.sState := 'unknown';
	END_CASE
	
(* End *)
END_ACTION

ACTION act_DiagObjectsBits:
(* act_TsDiagObjectsBits *)

	stTsSlaveInfo.stTsDiagObjectsBitsEL1904.bErrInput1		 			 := stDiagObjects.nSensorTestError.0;
	stTsSlaveInfo.stTsDiagObjectsBitsEL1904.bErrInput2		 			 := stDiagObjects.nSensorTestError.1;
	stTsSlaveInfo.stTsDiagObjectsBitsEL1904.bErrInput3		 			 := stDiagObjects.nSensorTestError.2;
	stTsSlaveInfo.stTsDiagObjectsBitsEL1904.bErrInput4		 			 := stDiagObjects.nSensorTestError.1;
	
	stTsSlaveInfo.stTsDiagObjectsBitsEL1904.bErrFirstInputPair 			 := stDiagObjects.nDuringTwoChannelEvaluationError.0;
	stTsSlaveInfo.stTsDiagObjectsBitsEL1904.bErrSecondInputPair 		 := stDiagObjects.nDuringTwoChannelEvaluationError.1;

	stTsSlaveInfo.stTsDiagObjectsBitsEL1904.bMatOpModeErrFirstInputPair	 := stDiagObjects.nMatModeInputPairDisagreeError.0 
																				AND stDiagObjects.nMatModeInputPairDisagreeError.1;
	stTsSlaveInfo.stTsDiagObjectsBitsEL1904.bMatOpModeErrSecondInputPair := stDiagObjects.nMatModeInputPairDisagreeError.2 
																				AND stDiagObjects.nMatModeInputPairDisagreeError.3;

	stTsSlaveInfo.stTsDiagObjectsBitsEL1904.bMatOpModeExtSupplyErrInput1 := stDiagObjects.nMatModeExternalSupplyError.0;
	stTsSlaveInfo.stTsDiagObjectsBitsEL1904.bMatOpModeExtSupplyErrInput2 := stDiagObjects.nMatModeExternalSupplyError.1;
	stTsSlaveInfo.stTsDiagObjectsBitsEL1904.bMatOpModeExtSupplyErrInput3 := stDiagObjects.nMatModeExternalSupplyError.2;
	stTsSlaveInfo.stTsDiagObjectsBitsEL1904.bMatOpModeExtSupplyErrInput4 := stDiagObjects.nMatModeExternalSupplyError.3;

(* End *)
END_ACTION

ACTION act_EcSlaveIdentify:
(* Identify the EtherCAT slave *)

	IF NOT nEcSlaveState.3
	THEN
		stTsSlaveInfo.bSlaveIdentify  	   := FALSE;
		stTsSlaveInfo.bSlaveTypeError 	   := FALSE;
		stTsSlaveInfo.sEcSlaveType         := '';
		stTsSlaveInfo.bSlaveAddressOk 	   := FALSE;
		stTsSlaveInfo.nEcSlaveFSoEAddr 	   := 0;
		stTsSlaveInfo.nEcSlaveSerialNumber := 0;
	END_IF

	IF nEcSlaveState.3
		AND NOT stTsSlaveInfo.bSlaveIdentify
		AND NOT stTsSlaveInfo.bSlaveTypeError
 		AND F_CreateAmsNetId(stEcAdsAddr.netId) <> '0.0.0.0.0.0' 
		AND stEcAdsAddr.port <> 0
	THEN

		fbEcCoeSdoRead(
			sNetId			:= 	F_CreateAmsNetId(stEcAdsAddr.netId),
			nSlaveAddr		:= 	stEcAdsAddr.port,
			nSubIndex		:= 	0,
			nIndex			:= 	16#1008,
			pDstBuf			:= 	ADR(stTsSlaveInfo.sEcSlaveType),
			cbBufLen		:= 	SIZEOF(stTsSlaveInfo.sEcSlaveType),
			bExecute		:= 	TRUE,
			tTimeout		:= 	DEFAULT_ADS_TIMEOUT);
	

		fbEcGetSlaveName(
			bExecute		:=	TRUE, 
			sNetId			:=	F_CreateAmsNetId(stEcAdsAddr.netId), 
			nSlaveAddr		:=	stEcAdsAddr.port, 
			tTimeout		:=	DEFAULT_ADS_TIMEOUT, 
			bBusy			=>	, 
			sSlaveName		=>	stTsSlaveInfo.sEcSlaveName, 
			bError			=>	, 
			nErrId			=>	);

		IF NOT fbEcCoeSdoRead.bBusy
			AND NOT fbEcCoeSdoRead.bError
			AND NOT fbEcGetSlaveName.bBusy
			AND NOT fbEcGetSlaveName.bError
		THEN

			fbEcCoeSdoRead(bExecute := FALSE); 
			fbEcGetSlaveName(bExecute := FALSE); 

			IF stTsSlaveInfo.sEcSlaveType = 'EL1904' 
				AND fbEcGetSlaveName.sSlaveName <> ''
			THEN
				stTsSlaveInfo.bSlaveIdentify := TRUE;
			ELSE
				stTsSlaveInfo.bSlaveTypeError := TRUE;
			END_IF

		ELSIF NOT fbEcCoeSdoRead.bBusy
			AND fbEcCoeSdoRead.bError
		OR (NOT fbEcGetSlaveName.bBusy
			AND fbEcGetSlaveName.bError)
		THEN
		
			fbEcCoeSdoRead  (bExecute := FALSE); 
			fbEcGetSlaveName(bExecute := FALSE); 

		END_IF

	END_IF
	

	IF nEcSlaveState.3
		AND stTsSlaveInfo.bSlaveIdentify
			AND NOT stTsSlaveInfo.bSlaveAddressOk
	THEN
		// Read slave FSoE Address  (F980:01)
		// Read slave serial number (F980:02)

			fbEcCoeSdoRead(
				sNetId			:= 	F_CreateAmsNetId(stEcAdsAddr.netId),
				nSlaveAddr		:= 	stEcAdsAddr.port,
				nSubIndex		:= 	1,
				nIndex			:= 	16#F980,
				pDstBuf			:= 	ADR(stTsSlaveInfo.stTsSlaveAddress),
				cbBufLen		:= 	SIZEOF(stTsSlaveInfo.stTsSlaveAddress),
				bExecute		:= 	TRUE,
				tTimeout		:= 	DEFAULT_ADS_TIMEOUT,
				bCompleteAccess	:= 	TRUE);

			IF NOT fbEcCoeSdoRead.bBusy 
				AND NOT fbEcCoeSdoRead.bError 
			THEN
				fbEcCoeSdoRead(bExecute := FALSE);
				stTsSlaveInfo.nEcSlaveFSoEAddr 		:= stTsSlaveInfo.stTsSlaveAddress.nEcSlaveFSoEAddr;
				stTsSlaveInfo.nEcSlaveSerialNumber 	:= TO_UDINT(stTsSlaveInfo.stTsSlaveAddress.nEcSlaveSerialNumber[0] OR SHL(TO_DWORD(stTsSlaveInfo.stTsSlaveAddress.nEcSlaveSerialNumber[1]),16));
				stTsSlaveInfo.bSlaveAddressOk 		:= TRUE;
			ELSIF NOT fbEcCoeSdoRead.bBusy 
				AND fbEcCoeSdoRead.bError 
			THEN
				fbEcCoeSdoRead(bExecute := FALSE);
				stTsSlaveInfo.nEcSlaveFSoEAddr 		:= 0;
				stTsSlaveInfo.nEcSlaveSerialNumber 	:= 0;
			END_IF	
	
	END_IF
	
(* End *)
END_ACTION

ACTION act_ReadDiagObjects:
(* Evaluate the Terminal temperatures and diagnostic objects *)

	CASE eReadDiagObjState OF

		eCycleDiagObj_Init				:	(* Init *)	

			IF nEcSlaveState.3					(* Slave in OP *)
				AND tCoEReadCycle <> T#0MS 		(* tCoEReadCycle <> t#0ms -> Read diagnostic aktiv *)
			THEN
				bReadDiagObjError := FALSE;
				fbEcCoeSdoRead(	bExecute := FALSE);
				fbTimer(IN := FALSE);
				eReadDiagObjState := eCycleDiagObj_ReadTemperature;
			END_IF

			
		eCycleDiagObj_ReadTemperature	:	(* Read temperature *)

			fbEcCoeSdoRead(
				sNetId			:= 	F_CreateAmsNetId(stEcAdsAddr.netId),
				nSlaveAddr		:= 	stEcAdsAddr.port,
				nSubIndex		:= 	1,
				nIndex			:= 	16#FA80,
				pDstBuf			:= 	ADR(stTsSlaveInfo.stSlaveTemp),
				cbBufLen		:= 	SIZEOF(stTsSlaveInfo.stSlaveTemp),
				bExecute		:= 	TRUE,
				tTimeout		:= 	DEFAULT_ADS_TIMEOUT,
				bCompleteAccess	:= 	TRUE);

			IF NOT fbEcCoeSdoRead.bBusy 
				AND NOT fbEcCoeSdoRead.bError 
			THEN
				fbEcCoeSdoRead(bExecute := FALSE);
				eReadDiagObjState := eCycleDiagObj_ReadDiag;
			ELSIF NOT fbEcCoeSdoRead.bBusy 
				AND fbEcCoeSdoRead.bError 
			THEN
				eReadDiagObjErrStep := eReadDiagObjState;
				eReadDiagObjState 	:= eCycleDiagObj_Error;
			END_IF

			
		eCycleDiagObj_ReadDiag			:	(* Read diacnostic objects *)

			fbTimer(IN := TRUE, PT := tCoEReadCycle);

			fbEcCoeSdoRead(
				sNetId			:= 	F_CreateAmsNetId(stEcAdsAddr.netId),
				nSlaveAddr		:= 	stEcAdsAddr.port,
				nSubIndex		:= 	1,
				nIndex			:= 	16#800E,
				pDstBuf			:= 	ADR(stDiagObjects),
				cbBufLen		:= 	SIZEOF(stDiagObjects),
				bExecute		:= 	TRUE,
				tTimeout		:= 	DEFAULT_ADS_TIMEOUT,
				bCompleteAccess	:= 	TRUE);

			IF NOT fbEcCoeSdoRead.bBusy 
				AND NOT fbEcCoeSdoRead.bError 
			THEN
				fbEcCoeSdoRead(bExecute := FALSE);
				act_DiagObjectsBits();
				eReadDiagObjState := eCycleDiagObj_ReadDelay;
			ELSIF NOT fbEcCoeSdoRead.bBusy 
				AND fbEcCoeSdoRead.bError 
			THEN
				eReadDiagObjErrStep := eReadDiagObjState;
				eReadDiagObjState 	:= eCycleDiagObj_Error;
			END_IF
				
			
		eCycleDiagObj_ReadDelay		:	(* Read delay *)
			fbTimer(
				IN := TRUE, 
				PT := tCoEReadCycle);

			IF fbTimer.Q 
			THEN
				fbTimer(IN := FALSE); 			
				eReadDiagObjState := eCycleDiagObj_Done;
			END_IF

			
		eCycleDiagObj_Done				:	(* Done *)

			eReadDiagObjState := eCycleDiagObj_Init;

			
		eCycleDiagObj_Error			:	(* Error detected *)

			bReadDiagObjError := TRUE;
		
			IF bReadDiagObjReset
			THEN
				bReadDiagObjError := FALSE;
				fbEcCoeSdoRead(bExecute := FALSE);
				eReadDiagObjErrStep := E_TsCycleDiagObj.eCycleDiagObj_NoError;
				eReadDiagObjState := eCycleDiagObj_Init;
			END_IF

	ELSE
		
		eReadDiagObjState := eCycleDiagObj_Init;
		
	END_CASE

	stTsSlaveInfo.bIntTempWarning1 := stTsSlaveInfo.stSlaveTemp.nInternalTemperature1 >= nWarningLevelTemp1;
	stTsSlaveInfo.bIntTempWarning2 := stTsSlaveInfo.stSlaveTemp.nInternalTemperature2 >= nWarningLevelTemp2;
									
(* End *)
END_ACTION

ACTION act_Signals:
(* Evaluate the input (EL1904) signals *)

	IF nEcSlaveState.3 (* Slave in operational state *)
	THEN
		(* OP -> transfer the signal states *)
		stTsSlaveInfo.bChannel1 := stInfoData.nInOutSafeDataByte1.0;
		stTsSlaveInfo.bChannel2 := stInfoData.nInOutSafeDataByte1.1;
		stTsSlaveInfo.bChannel3 := stInfoData.nInOutSafeDataByte1.2;
		stTsSlaveInfo.bChannel4 := stInfoData.nInOutSafeDataByte1.3;
	ELSE
		(* Error -> clear the signal states *)
		stTsSlaveInfo.bChannel1 := FALSE; 
		stTsSlaveInfo.bChannel2 := FALSE;
		stTsSlaveInfo.bChannel3 := FALSE; 
		stTsSlaveInfo.bChannel4 := FALSE;
	END_IF

(* End *)
END_ACTION

END_FUNCTION_BLOCK

// ---- POUs/FB_TwinSafeFB.TcPOU
FUNCTION_BLOCK FB_TwinSafeFB
(*******************************************************************************************************
Description			:	Entries of the status and diagnostic TwinSAFE function blocks
Documentation 		:	TwinSAFE-Logik-FB TwinCAT function blocks for TwinSAFE logic terminals
Supported hardware	: 	KL6904 / EL6900 / EL6910 / EJ6910 / EK1960
Version/Date 		:	V3.1.0/26.10.2016
********************************************************************************************************)
VAR_INPUT

	sName									:STRING;		(* TwinSAFE function block Name in the TwinSAFE project *)
	eFBType									:E_TsFbType;	(* TwinSAFE function block type in the TwinSAFE project *)
	nFbId									:UINT;			(* TwinSAFE function block ID in the TwinSAFE project *)

END_VAR
VAR_OUTPUT
	
	stInfoData						AT%I* 	:ST_TsFbInfo;	(* Function Block Info Data *)
	sType									:STRING;
	sState									:STRING;
	sDiag									:STRING;

END_VAR
VAR
END_VAR
(* End *)

(* TwinSAFE function block status and diagnosis *)	

(* THIS CODE IS ONLY AN EXAMPLE - YOU HAVE TO CHECK APTITUDE FOR YOUR APPLICATION *)

	CASE eFBType OF
		
		FB_TYPE_AND					:	(* TwinSAFE function block - AND *)

			sType := 'AND';
			
			CASE stInfoData.nState OF
				1:		sState := 'RUN';	
				2:		sState := 'STOP';	
				3:		sState := 'SAFE';	
			ELSE 
				sState := 'undefined';
			END_CASE
			
			sDiag := 'NOT IN USE';


		FB_TYPE_OR					:	(* TwinSAFE function block - OR *)

			sType := 'OR';
			
			CASE stInfoData.nState OF
				1:		sState := 'RUN';	
				2:		sState := 'STOP';	
				3:		sState := 'SAFE';	
			ELSE 	
				sState := 'undefined';
			END_CASE

			sDiag := 'NOT IN USE';

			
		FB_TYPE_OPMODE				:	(* TwinSAFE function block - OPMODE *)

			sType := 'OPMODE';
			
			CASE stInfoData.nState OF
				1:		sState := 'RUN';	
				2:		sState := 'STOP';	
				3:		sState := 'SAFE';	
				4:		sState := 'ERROR';	
				5:		sState := 'RESET';	
				6:		sState := 'START';	
			ELSE 
				sState := 'undefined';
			END_CASE
			
			CASE stInfoData.nDiag OF
				0:	sDiag := 'No error';		
				1:	sDiag := 'Discrepancy monitoring error';		
			ELSE 
				sDiag := 'undefined';
			END_CASE


		FB_TYPE_ESTOP				:	(* TwinSAFE function block - ESTOP *)

			sType := 'ESTOP';
			
			CASE stInfoData.nState OF
				1:		sState := 'RUN';	
				2:		sState := 'STOP';	
				3:		sState := 'SAFE';	
				4:		sState := 'ERROR';	
				5:		sState := 'RESET';	
				6:		sState := 'START';	
				8:		sState := 'DELAYOUT';	
			ELSE 
				sState := 'undefined';
			END_CASE

			
			sDiag := '';
			
			CASE TO_WORD(stInfoData.nDiag) AND 16#00FF OF
				1:		sDiag := 'Discrepancy error input group 1';
				2:		sDiag := 'Discrepancy error input group 2';
				4:		sDiag := 'Discrepancy error input group 3';
				8:		sDiag := 'Discrepancy error input group 4';
				16:		sDiag := 'EDM monitoring error EDM1';
				32:		sDiag := 'EDM monitoring error EDM2';
			END_CASE

			CASE TO_WORD(stInfoData.nDiag) AND 16#FF00 OF
				256:	sDiag := CONCAT(sDiag, ' - option "SAFE Inputs after Disc Error" aktiv');
				512:	sDiag := CONCAT(sDiag, ' - option "SAFE Inputs after Disc Error" aktiv');
				1024:	sDiag := CONCAT(sDiag, ' - option "SAFE Inputs after Disc Error" aktiv');
				2048:	sDiag := CONCAT(sDiag, ' - option "SAFE Inputs after Disc Error" aktiv');
			END_CASE
				
			IF stInfoData.nDiag = 0
			THEN
				sDiag := 'No error';
			ELSIF sDiag = ''
			THEN
				sDiag := 'undefined';		
			END_IF

			
		FB_TYPE_MON					:	(* TwinSAFE function block - MON *)

			sType := 'MON';
			
			CASE stInfoData.nState OF
				1:		sState := 'RUN';	
				2:		sState := 'STOP';	
				3:		sState := 'SAFE';	
				4:		sState := 'ERROR';	
				5:		sState := 'RESET';	
				6:		sState := 'START';	
				7:		sState := 'ERRORDELAY';	
				8:		sState := 'DELAYOUT';	
				9:		sState := 'FUNCTEST';	
			ELSE 
				sState := 'undefined';
			END_CASE
			
			CASE stInfoData.nDiag OF
				0:		sDiag := 'No error';		
				1:		sDiag := 'Discrepancy error input group 1';	
				2:		sDiag := 'Discrepancy error input group 1';		
				4:		sDiag := 'Discrepancy error in Secure input group';	
				16:		sDiag := 'EDM monitoring error EDM1';	
				32:		sDiag := 'EDM monitoring error EDM2';	
			ELSE 
				sDiag := 'undefined';
			END_CASE


		FB_TYPE_DECOUPLER			:	(* TwinSAFE function block - DECOUPLER *)

			sType := 'DECOUPLER';
			
			CASE stInfoData.nState OF
				1:		sState := 'RUN';	
				2:		sState := 'STOP';	
			ELSE 
				sState := 'undefined';
			END_CASE

			sDiag := 'NOT IN USE';

			
		FB_TYPE_TWOHAND				:	(* TwinSAFE function block - TWOHAND *)

			sType := 'TWO-HAND';
			
			CASE stInfoData.nState OF
				1:		sState := 'RUN';	
				2:		sState := 'STOP';	
				3:		sState := 'SAFE';	
				4:		sState := 'ERROR';		
				5:		sState := 'RESET';	
				6:		sState := 'START';	
				11:		sState := '1BUTTON';	
				12:		sState := '2BUTTON';	
				13:		sState := 'RELEASE';	
			ELSE 
				sState := 'undefined';
			END_CASE
			
			CASE stInfoData.nDiag OF
				0:		sDiag := 'No error';		
				1:		sDiag := 'Discrepancy error input group 1';	
				2:		sDiag := 'Discrepancy error input group 1';	
				4:		sDiag := 'Discrepancy error between the two input groups';	
				64:		sDiag := 'Two-hand error';	
			ELSE 
				sDiag := 'undefined';
			END_CASE

	
		FB_TYPE_MUTING				:	(* TwinSAFE function block - MUTING  *)

			sType := 'MUTING';
			
			CASE stInfoData.nState OF
				1:		sState := 'RUN';	
				2:		sState := 'STOP';	
				3:		sState := 'SAFE';	
				4:		sState := 'ERROR';	
				5:		sState := 'RESET';	
				8:		sState := 'DELAYOUT';	
				9:		sState := 'MUTING1';	
				10:		sState := 'MUTING2';	
				11:		sState := 'MUTING3';	
				12:		sState := 'MUTING4';	
				13:		sState := 'MUTING5';	
				14:		sState := 'MUTING6';	
				15:		sState := 'MUTING7';	
				16:		sState := 'MUTING8';	
				17:		sState := 'MUTING9';	
			ELSE 
				sState := 'undefined';
			END_CASE
			
			CASE stInfoData.nDiag OF
				0:		sDiag := 'No error';		
				1:		sDiag := 'Discrepancy error in muting input group 1';	
				2:		sDiag := 'Discrepancy error in the OSSD input group';	
				4:		sDiag := 'Discrepancy error in muting input group 2';	
				16:		sDiag := 'EDM monitoring error EDM1';	
				32:		sDiag := 'EDM monitoring error EDM2';	
				64:		sDiag := 'Muting sequence was violated';	
				128:	sDiag := 'Maximum muting time was exceeded';	
			ELSE 
				sDiag := 'undefined';
			END_CASE

		
		FB_TYPE_EDM					:	(* TwinSAFE function block - EDM *)

			sType := 'EDM';
			
			CASE stInfoData.nState OF
				2:		sState := 'STOP';	
				4:		sState := 'ERROR';	
				5:		sState := 'RESET';	
				14:		sState := 'MON_OFF';	
				15:		sState := 'MON_ON';	
			ELSE 
				sState := 'undefined';
			END_CASE
			
			CASE stInfoData.nDiag OF
				0:		sDiag := 'No error';		
				1:		sDiag := 'Switch-OFF timer elapsed';	
				2:		sDiag := 'Switch-ON timer elapsed';	
			ELSE 
				sDiag := 'undefined';
			END_CASE

			
		FB_TYPE_RS					:	(* TwinSAFE function block - RS *)

			sType := 'RS';

			CASE stInfoData.nState OF
				2:		sState := 'STOP';	
				3:		sState := 'SAFE';	
				9:		sState := 'SET';	
			ELSE 
				sState := 'undefined';
			END_CASE

			sDiag := 'NOT IN USE';


		FB_TYPE_SR					:	(* TwinSAFE function block - SR *)

			sType := 'SR';
			
			CASE stInfoData.nState OF
				2:		sState := 'STOP';	
				3:		sState := 'SAFE';	
				9:		sState := 'SET';	
			ELSE 
				sState := 'undefined';
			END_CASE
			
			sDiag := 'NOT IN USE';
	

		FB_TYPE_TON					:	(* TwinSAFE function block - TON *)

			sType := 'TON';
			
			CASE stInfoData.nState OF
				1:		sState := 'RUN';	
				2:		sState := 'STOP';	
				3:		sState := 'SAFE';	
				9:		sState := 'DELAY_IN';	
			ELSE 
				sState := 'undefined';
			END_CASE

			sDiag := 'NOT IN USE';


		FB_TYPE_TOF					:	(* TwinSAFE function block - TOF *)

			sType := 'TOF';
			
			CASE stInfoData.nState OF
				1:		sState := 'RUN';	
				2:		sState := 'STOP';	
				3:		sState := 'SAFE';	
				8:		sState := 'DELAY_OUT';	
			ELSE 
				sState := 'undefined';
			END_CASE

			sDiag := 'NOT IN USE';


		FB_TYPE_CONSHUT				:	(* TwinSAFE function block - CONNECTION SHUTDOWN *)

			sType := 'ConShut';
			
			CASE stInfoData.nState OF
				2:		sState := 'STOP';	
				3:		sState := 'SAFE';	
				4:		sState := 'ERROR';	
				5:		sState := 'RESET';	
				10:		sState := 'ACTIVE';	
				11:		sState := 'DEACTIVE';	
			ELSE 
				sState := 'undefined';
			END_CASE
			
			CASE stInfoData.nDiag OF
				0:		sDiag := 'No error';		
				1:		sDiag := 'Discrepancy error input group 1';	
			ELSE 
				sDiag := 'undefined';
			END_CASE
			
			
		FB_TYPE_ADD					:	(* TwinSAFE function block - ADD *)

			sType := 'ADD';
			
			CASE stInfoData.nState OF
				0:		sState := 'not in use';	
				1:		sState := 'RUN';	
				2:		sState := 'STOP';	
				3:		sState := 'not in use';	
				4:		sState := 'ERROR';	
				5:		sState := 'RESET';	
			ELSE 
				sState := 'undefined';
			END_CASE

			CASE stInfoData.nDiag OF
				0:		sDiag := 'AnalogOut is correct';		
				1:		sDiag := 'AnalogOut has an underflow';	
				2:		sDiag := 'AnalogOut has an overflow';	
			ELSE 
				sDiag := 'undefined';
			END_CASE
			
			
		FB_TYPE_SUB					:	(* TwinSAFE function block - SUB *)

			sType := 'SUB';
			
			CASE stInfoData.nState OF
				0:		sState := 'not in use';	
				1:		sState := 'RUN';	
				2:		sState := 'STOP';	
				3:		sState := 'not in use';	
				4:		sState := 'ERROR';	
				5:		sState := 'RESET';	
			ELSE 
				sState := 'undefined';
			END_CASE

			CASE stInfoData.nDiag OF
				0:		sDiag := 'AnalogOut is correct';		
				1:		sDiag := 'AnalogOut has an underflow';	
				2:		sDiag := 'AnalogOut has an overflow';	
			ELSE 
				sDiag := 'undefined';
			END_CASE

			
		FB_TYPE_MUL					:	(* TwinSAFE function block - MUL *)

			sType := 'MUL';
			
			CASE stInfoData.nState OF
				0:		sState := 'not in use';	
				1:		sState := 'RUN';	
				2:		sState := 'STOP';	
				3:		sState := 'not in use';	
				4:		sState := 'ERROR';	
				5:		sState := 'RESET';	
			ELSE 
				sState := 'undefined';
			END_CASE

			CASE stInfoData.nDiag OF
				0:		sDiag := 'AnalogOut is correct';		
				1:		sDiag := 'AnalogOut has an underflow';	
				2:		sDiag := 'AnalogOut has an overflow';	
			ELSE 
				sDiag := 'undefined';
			END_CASE

			
		FB_TYPE_DIV					:	(* TwinSAFE function block - DIV *)

			sType := 'DIV';
			
			CASE stInfoData.nState OF
				0:		sState := 'not in use';	
				1:		sState := 'RUN';	
				2:		sState := 'STOP';	
				3:		sState := 'not in use';	
				4:		sState := 'ERROR';	
				5:		sState := 'RESET';	
			ELSE 
				sState := 'undefined';
			END_CASE

			CASE stInfoData.nDiag OF
				0:		sDiag := 'AnalogOut is correct';		
				1:		sDiag := 'AnalogOut has an underflow';	
				2:		sDiag := 'AnalogOut has an overflow';	
			ELSE 
				sDiag := 'undefined';
			END_CASE


		FB_TYPE_COMPARE				:	(* TwinSAFE function block - COMPARE *)

			sType := 'COMPARE';
			
			CASE stInfoData.nState OF
				1:		sState := 'RUN';	
				2:		sState := 'STOP';	
				3:		sState := 'SAFE';	
				4:		sState := 'ERROR';	
				5:		sState := 'RESET';	
				8:		sState := 'DELAYOUT';	
			ELSE 
				sState := 'undefined';
			END_CASE

			CASE stInfoData.nDiag OF
				0:		sDiag := 'CompOut is correct';		
				1:		sDiag := 'The output CompOut has an underflow';	
				2:		sDiag := 'The output CompOut has an overflow';	
			ELSE 
				sDiag := 'undefined';
			END_CASE
			
			
		FB_TYPE_LIMIT				:	(* TwinSAFE function block - LIMIT *)

			sType := 'LIMIT';
			
			CASE stInfoData.nState OF
				1:		sState := 'RUN';	
				2:		sState := 'STOP';	
				3:		sState := 'SAFE';	
				4:		sState := 'ERROR';	
				5:		sState := 'RESET';	
			ELSE 
				sState := 'undefined';
			END_CASE

			CASE stInfoData.nDiag OF
				0:		sDiag := 'No error';		
				1:		sDiag := 'MinValue > MaxValue';	
			ELSE 
				sDiag := 'undefined';
			END_CASE
			
			
		FB_TYPE_COUNTER				:	(* TwinSAFE function block - COUNTER *)

			sType := 'COUNTER';
			
			CASE stInfoData.nState OF
				1:		sState := 'RUN';	
				2:		sState := 'STOP';	
				4:		sState := 'ERROR';	
				5:		sState := 'RESET';	
			ELSE 
				sState := 'undefined';
			END_CASE

			CASE stInfoData.nDiag OF
				0:		sDiag := 'No error';		
				1:		sDiag := 'ActValue has an underflow';	
				2:		sDiag := 'ActValue has an overflow';	
			ELSE 
				sDiag := 'undefined';
			END_CASE


		FB_TYPE_SCALE				:	(* TwinSAFE function block - SCALE *)

			sType := 'SCALE';
			
			CASE stInfoData.nState OF
				1:		sState := 'RUN';	
				2:		sState := 'STOP';	
				4:		sState := 'ERROR';	
				5:		sState := 'RESET';	
			ELSE 
				sState := 'undefined';
			END_CASE

			CASE stInfoData.nDiag OF
				0:		sDiag := 'No error';		
				1:		sDiag := 'AnalogOut has an underflow';	
				2:		sDiag := 'AnalogOut has an overflow';	
				3:		sDiag := 'A 32-bit overflow occurs during the multiplication';	
				4:		sDiag := 'A 32-bit overflow occurs during by rounding up at the division ';	
			ELSE 
				sDiag := 'undefined';
			END_CASE


		FB_TYPE_SPEED				:	(* TwinSAFE function block - SPEED *)

			sType := 'SPEED';
			
			CASE stInfoData.nState OF
				1:		sState := 'RUN';	
				2:		sState := 'STOP';	
				4:		sState := 'ERROR';	
				5:		sState := 'RESET';	
			ELSE 
				sState := 'undefined';
			END_CASE

			CASE stInfoData.nDiag OF
				0:		sDiag := 'No error';		
				1:		sDiag := 'The output Speed has an underflow';	
				2:		sDiag := 'The output Speed has an overflow';	
			ELSE 
				sDiag := 'undefined';
			END_CASE


		FB_TYPE_LOADSENSING			:	(* TwinSAFE function block - LOAD SENSING *)

			sType := 'LOADSENSING';
			
			CASE stInfoData.nState OF
				1:		sState := 'RUN';	
				2:		sState := 'STOP';	
				3:		sState := 'SAFE';	
				16:		sState := 'INACTIVE';	
				17:		sState := 'WARNING';	
			ELSE 
				sState := 'undefined';
			END_CASE

			sDiag := 'NOT IN USE';


		FB_TYPE_CAMMONITOR			:	(* TwinSAFE function block - CAM MONITOR *)

			sType := 'CAMMONITOR';
			
			CASE stInfoData.nState OF
				1:		sState := 'RUN';	
				2:		sState := 'STOP';	
				3:		sState := 'SAFE';	
				4:		sState := 'ERROR';	
				5:		sState := 'RESET';	
				6:		sState := 'START';	
				15:		sState := 'WAIT-FOR-RESET';	
				16:		sState := 'MOVE-STOP';	
				17:		sState := 'MOVE-START';	
				18:		sState := 'MOVE-DOWN';	
				19:		sState := 'MOVE-UP';	
				20:		sState := 'MOVE-TDC';	
				32:		sState := 'MOVE-DOWN-CLOCKWISE';	
				33:		sState := 'MOVE-UP-CLOCKWISE';	
				34:		sState := 'MOVE-UP-TDC1';	
				35:		sState := 'MOVE-STOP-TDC1';	
				36:		sState := 'MOVE-START-TDC1';	
				37:		sState := 'MOVE-DOWN-CONTRA-CLOCKWISE';	
				38:		sState := 'MOVE-UP-CONTRA-CLOCKWISE';	
				39:		sState := 'MOVE-UP-TDC2';	
				40:		sState := 'MOVE-STOP-TDC2';	
				41:		sState := 'MOVE-START-TDC2';	
			ELSE 
				sState := 'undefined';
			END_CASE

			sDiag := 'NOT IN USE';


		FB_TYPE_SLI					:	(* TwinSAFE function block - SLI *)

			sType := 'SLI';
			
			CASE stInfoData.nState OF
				1:		sState := 'RUN';	
				2:		sState := 'STOP';	
				3:		sState := 'SAFE';	
				4:		sState := 'ERROR';	
				5:		sState := 'RESET';	
			ELSE 
				sState := 'undefined';
			END_CASE

			CASE stInfoData.nDiag OF
				0:		sDiag := 'No error';		
				1:		sDiag := 'Underflow (PositionDiff < -NegLimit)';		
				2:		sDiag := 'Overflow (PositionDiff > PosLimit)';		
			ELSE 
				sDiag := 'undefined';
			END_CASE


		FB_TYPE_ENVELOPE			:	(* TwinSAFE function block - ENVELOPE *)

			sType := 'ENVELOPE';
			
			CASE stInfoData.nState OF
				1:		sState := 'RUN';	
				2:		sState := 'STOP';	
				3:		sState := 'SAFE';	
				4:		sState := 'ERROR';	
				5:		sState := 'RESET';	
				8:		sState := 'DELAYOUT';	
				9:		sState := 'MONITOR';	
			ELSE 
				sState := 'undefined';
			END_CASE

			CASE stInfoData.nDiag OF
				0:		sDiag := 'No error';		
				1:		sDiag := 'Underflow (InValue below the envelope curve)';		
				2:		sDiag := 'Overflow (InValue above the envelope curve)';		
				3:		sDiag := 'InValue error';		
				4:		sDiag := 'Max time expired)';		
			ELSE 
				sDiag := 'undefined';
			END_CASE


		FB_TYPE_VIOLATIONCOUNTER	:	(* TwinSAFE function block - VIOLATION COUNTER *)

			sType := 'VIOLATIONCOUNTER';
			
			CASE stInfoData.nState OF
				1:		sState := 'RUN';	
				2:		sState := 'STOP';	
				3:		sState := 'SAFE';	
				6:		sState := 'START';	
			ELSE 
				sState := 'undefined';
			END_CASE

			sDiag := 'NOT IN USE';


	ELSE
		
		sType  := 'UNKNOWN FB';
		sState := 'UNKNOWN';
		sDiag  := 'UNKNOWN';

	END_CASE
	
	sType := CONCAT(' : ', sType);
	sType := CONCAT(UINT_TO_STRING(nFbId), sType);
	sType := CONCAT('FB ', sType);
	
(* End *)

END_FUNCTION_BLOCK

// ---- POUs/F_Scale.TcPOU
FUNCTION F_Scale : INT
VAR_INPUT
	nAIn: DINT;
	fOutMin: REAL; // Maximum of the output value
	fOutMax: REAL; // Minimum of the output value
	nInMin: DINT; // Minimum of the input value
	nInMax: DINT; // Maximum of the input value
END_VAR
VAR
	fAIn: REAL;
	fSlope: REAL;
	fConstant: REAL;
	fInMax: REAL;
	fInMin: REAL;
END_VAR

// Binding rules
IF nAIn >= nInMax THEN
	nAIN := nInMax;
ELSIF nAIn <= nInMin THEN
	nAIn := nInMin;
END_IF

fAIn := DINT_TO_REAL(nAIn);
fInMax := DINT_TO_REAL(nInMax);
fInMin := DINT_TO_REAL(nInMin);

// y = ax + b

// Find a
fSlope := (fOutMax-fOutMin)/(fInMax-fInMin);

// Find b
fConstant := fOutMin - (fSlope * fInMin);

F_Scale := REAL_TO_INT(fSlope*fAin + fConstant);

END_FUNCTION

// ---- POUs/FB_TwinSafeGroup.TcPOU
FUNCTION_BLOCK FB_TwinSafeGroup
(*******************************************************************************************************
Description			:	Entries of the status and diagnostic TwinSAFE groups
ocumentation 		:	TwinSAFE-Logik-FB TwinCAT function blocks for TwinSAFE logic terminals
Supported hardware	: 	KL6904 / EL6900
Version/Date 		:	V3.1.0/26.10.2016
********************************************************************************************************)
VAR_INPUT

	bRun							AT %Q*	:BOOL;				(* TwinSAFE group run - linked with the associated TwinSAFE Group in the TwinSAFE projekt *)
	bErrAck							AT %Q*	:BOOL;				(* TwinSAFE group error acknowledge - linked with the associated TwinSAFE Group in the TwinSAFE projekt *)
	sName									:STRING;			(* TwinSAFE group name *)

END_VAR
VAR_OUTPUT

	stInfoData						AT %I*	:ST_TsGroupInfo;	(* TwinSAFE Group Info Data *)
	bFbErr							AT %I*	:BOOL;				(* TwinSAFE group function block error - linked with the associated TwinSAFE Group in the TwinSAFE projekt *)
	bComErr							AT %I*	:BOOL;				(* TwinSAFE group communication error - linked with the associated TwinSAFE Group in the TwinSAFE projekt *)
	bOutErr							AT %I*	:BOOL;				(* TwinSAFE group output error - linked with the associated TwinSAFE Group in the TwinSAFE projekt *)
	sState									:STRING;
	
END_VAR
VAR
END_VAR
(* End *)

(* TwinSAFE group status and diagnostic *)

(* THIS CODE IS ONLY AN EXAMPLE - YOU HAVE TO CHECK APTITUDE FOR YOUR APPLICATION *)

	CASE stInfoData.nState OF
		1:	sState := 'RUN';
		2:	sState := 'STOP';
		3:	sState := 'SAFE';
		4:	sState := 'ERROR';
		5:	sState := 'RESET';
	ELSE
		sState := 'undefined';
	END_CASE

(* End *)

END_FUNCTION_BLOCK
